VAR_GLOBAL
	(* These global connection and namespace settings need to be adapted to the runtime environment *)
	(*sOpcUaServerUrl : STRING(MAX_STRING_LENGTH) := 'opc.tcp://localhost:4840';
	sNamespaceUri : STRING(MAX_STRING_LENGTH) := 'urn:BeckhoffAutomation:Ua:PLC1'; // TF6100 setup version 4.x default*)
	
	sOpcUaServerUrl : STRING(MAX_STRING_LENGTH) := 'opc.tcp://172.17.36.240:4840';
	sNamespaceUri : STRING(MAX_STRING_LENGTH) := 'urn:BeckhoffAutomation:Ua:PLC1'; // TF6100 setup version 4.x default
END_VAR

(* stored: Version 1.1.0.1, ProductVersion 3.1.4024.3
   GVL GlobalSettings: Id {eb05ed2f-70d2-4892-b1f1-f5dc3e9ac14b} *)
